# EPICS StreamDevice protocol: protocols/dio482_scaler.proto
Terminator = LF;
ExtraInput = Ignore;

get_dwell {
	out "dwell";
	in "%d";
}

set_dwell {
	out "dwell %d";
	in "";
}

get_acc {
	out "acc_not_reset";
	in "%d";
}

set_acc {
	out "acc_not_reset %d";
	in "";
}

get_cnt {
	out "cnt.\$1";
	in "%x";
}
